// This function has been automatically generated from the project information.
{attribute 'signature_flag' := '1073741824'}
{attribute 'TcGenerated'}
{attribute 'no-analysis'}
FUNCTION F_GetCompany : WSTRING
VAR_INPUT
	
END_VAR

F_GetCompany := "Kim Robbens";

END_FUNCTION

(* stored: Version 1.1.0.1
   POU F_GetCompany: Id {3eb07616-0567-4f53-abde-98b312a59f23}, SpecialFunc None *)
